PROGRAM MAIN
VAR
	I_StartButton: BOOL;
	I_StopButton: BOOL;
	Q_MotorRun: BOOL;
	tonContactor: TON;
	Q_Star: BOOL;
	Q_Delta: BOOL;
END_VAR

IF I_StartButton THEN
	Q_MotorRun := TRUE;
ELSIF I_StopButton THEN
	Q_MotorRun := FALSE;
END_IF

tonContactor(IN:= Q_MotorRun , PT:=T#10S);

Q_Star := Q_MotorRun AND NOT tonContactor.Q;
Q_Delta :=  Q_MotorRun AND NOT tonContactor.Q;

END_PROGRAM

(* stored: Version 1.1.0.1, ProductVersion 3.1.4024.9
   POU MAIN: Id {2b958d91-82b9-473c-805e-4eab70a71889}, SpecialFunc None *)
